SUBAPPLICATION mySubAppBlock (* Subapplication Type *)
  (* Standard: 61499-2 *)
  (* Version 1.0, 2025-07-11, dakudryashev *)
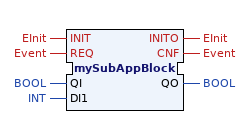
  EVENT_INPUT
    INIT : EInit; (* Initialization Request *)
    REQ; (* Normal Execution Request *)
  END_EVENT
  EVENT_OUTPUT
    INITO : EInit; (* Initialization Confirm *)
    CNF; (* Execution Confirmation *)
  END_EVENT
  VAR_INPUT
    QI : BOOL; (* Input event qualifier *)
    DI1 : INT;
  END_VAR
  VAR_OUTPUT
    QO : BOOL; (* Output event qualifier *)
  END_VAR
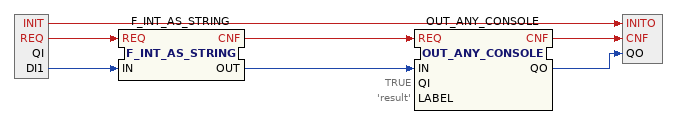
  FBS
    F_INT_AS_STRING : F_INT_AS_STRING;
    OUT_ANY_CONSOLE : OUT_ANY_CONSOLE(QI := TRUE, LABEL := 'result');
  END_FBS
  EVENT_CONNECTIONS
    REQ TO F_INT_AS_STRING.REQ;
    F_INT_AS_STRING.CNF TO OUT_ANY_CONSOLE.REQ;
    OUT_ANY_CONSOLE.CNF TO CNF;
    INIT TO INITO;
  END_CONNECTIONS
  DATA_CONNECTIONS
    DI1 TO F_INT_AS_STRING.IN;
    F_INT_AS_STRING.OUT TO OUT_ANY_CONSOLE.IN;
    OUT_ANY_CONSOLE.QO TO QO;
  END_CONNECTIONS
END_SUBAPPLICATION
